// ---- POUs/OperatingModes/MBS_OperatingModes.TcPOU
FUNCTION_BLOCK MBS_OperatingModes
VAR_INPUT
	Start 			: BOOL;
	Stop			: BOOL;
	Reset			: BOOL;
	Schalter		: BOOL;
	Schrittkette_GS : BOOL;
END_VAR
VAR_OUTPUT
	A1 : BOOL; //Initialzustand
	A2 : BOOL; //Stillstand angefordert am Ende des Zyklus
//	A3 : BOOL; //Stillstand angefordert in einem bestimmten Zustand
//	A4 : BOOL; //Erhaltener Stillstand
//	A5 : BOOL; //Vorbereitung zur Wiederaufnahme nach Störung
	A6 : BOOL; //Fahrt in den Initialzustand
	F1 : BOOL; //Normalbetrieb
//	F2 : BOOL; //Anfahren
//	F3 : BOOL; //Abfahren
	F4 : BOOL; //Handbetrieb
//	F5 : BOOL; //Schrittbetrieb
//	F6 : BOOL; //Testbetrieb
//	D1 : BOOL; //Not-Aus
//	D2 : BOOL; //DIagnose und Störbehandlung
//	D3 : BOOL; //Produktion trotz Störung
END_VAR
VAR
	bFirstScan : BOOL := TRUE;	
	
	RS_InitialState: RS;	
	RS_InitialDrive: RS;
	RS_ManualOperationMode: RS;
	RS_AutomaticOperationMode: RS;
	RS_CycleEnded: RS;

	R_TRIG_Manual: R_TRIG;
	R_TRIG_Automatic: R_TRIG;
	R_TRIG_InitialDrive: R_TRIG;
	R_TRIG_CycleEnded: R_TRIG;
	R_TRIG_Init: R_TRIG;
END_VAR

R_TRIG_InitialDrive(CLK := RS_InitialDrive);
R_TRIG_CycleEnded(CLK := RS_CycleEnded);
R_TRIG_Manual(CLK := RS_ManualOperationMode);
R_TRIG_Automatic(CLK := RS_AutomaticOperationMode);
RS_InitialState(SET := ((((R_TRIG_InitialDrive.Q) AND (Schrittkette_GS))) OR (((R_TRIG_CycleEnded.Q) AND (Schrittkette_GS)))), RESET1 := ((R_TRIG_Manual.Q) OR (R_TRIG_Automatic.Q)));
A1 := RS_InitialState.Q1;
RS_ManualOperationMode(SET := ((Schalter) AND (A1) AND (Reset)), RESET1 := A6);
F4 := RS_ManualOperationMode.Q1;
R_TRIG_Manual(CLK := RS_ManualOperationMode);
R_TRIG_Init(CLK := RS_InitialState);
RS_InitialDrive(SET := ((((R_TRIG_Manual.Q) AND (((Stop) OR (NOT (Schalter)))))) OR ((bFirstScan))), RESET1 := R_TRIG_Init.Q);
A6 := RS_InitialDrive.Q1;
R_TRIG_Init(CLK := RS_InitialState);
R_TRIG_CycleEnded(CLK := RS_CycleEnded);
RS_AutomaticOperationMode(SET := ((Start) AND (R_TRIG_Init.Q) AND (NOT (Schalter))), RESET1 := R_TRIG_CycleEnded.Q);
F1 := RS_AutomaticOperationMode.Q1;
R_TRIG_Automatic(CLK := RS_AutomaticOperationMode);
R_TRIG_Init(CLK := RS_InitialState);
RS_CycleEnded(SET := ((R_TRIG_Automatic.Q) AND (((Schalter) OR (Stop)))), RESET1 := R_TRIG_Init.Q);
A2 := RS_CycleEnded.Q1;

END_FUNCTION_BLOCK

// ---- POUs/MethodenBeispiele/FB_MyOpcUaMethod.TcPOU
FUNCTION_BLOCK PUBLIC FB_MyOpcUaMethod
VAR_INPUT
	in1 : INT;
	in2 : INT;
END_VAR
VAR_OUTPUT
	result : INT;
END_VAR

{attribute 'TcRpcEnable' := '1'}
METHOD PUBLIC Multiply : INT
VAR_INPUT
	a : INT;
	b : INT;
END_VAR
Multiply := a * b;
END_METHOD

END_FUNCTION_BLOCK

// ---- POUs/MethodenBeispiele/JobMethode_Schablone.TcPOU
{attribute 'OPC.UA.DA.JobMethod' := 'JobMethode_Schablone'}
FUNCTION_BLOCK JobMethode_Schablone
VAR
	AlwaysTrue : BOOL := TRUE;
	// Used for debugging purposes to display InputArguments of method call
	MethodCall_Name : BOOL := FALSE; // used to store InputArg "MethodCall" from Start() method
	Direction_01 : BOOL := FALSE;
	Direction_02 : BOOL := FALSE;
	TS_EndschalterEntlastung : BOOL;
	callCounterStart : ULINT; // counts how many times the Start() method has been called
	callCounterCheckState : ULINT; // counts how many times the CheckState() method has been called
	callCounterAbort : ULINT; // counts how many times the Abort() method has been called
	
	// Variables to determine if a job has been started (Start() method has been called) or finished
	jobRunning : BOOL;
	jobFinished : BOOL;

	// State machine variable
	state : UDINT;
	
	//Variablen des Transport FBs
	ResetCall : BOOL := FALSE;	
	JobMethode_Name : AxisControl_MultipleInputSensors;
END_VAR
	
VAR_INPUT
	NotAusSignal: BOOL;
	LightSensor_01 : BOOL;
	LightSensor_02 : BOOL;
	TS_Endschalter_01 : BOOL;
	TS_Endschalter_02 : BOOL;
	TOF_Time_Motoransteuerung : TIME;
	TOF_Time_EndschalterEntlastung : TIME;
END_VAR

VAR_OUTPUT
	Motor_Ansteuerung01 : BOOL;
	Motor_Ansteuerung02 : BOOL;
END_VAR

JobMethode_Name(
    MethodCall := MethodCall_Name,
    NotAus_Signal := NotAusSignal,
    Direction_01 := Direction_01,
    Direction_02 := Direction_02,
    LightSensor_01 := LightSensor_01,
    LightSensor_02 := LightSensor_02,
    TS_Endschalter_01 := TS_Endschalter_01,
    AutomaticMode := _REFACTOR_,
    TS_Endschalter_02 := TS_Endschalter_02,
    TS_EndschalterEntlastung := TS_EndschalterEntlastung,
    TOF_Time_Motoransteuerung := TOF_Time_Motoransteuerung,
    TOF_Time_EndschalterEntlastung := TOF_Time_EndschalterEntlastung
);
Motor_Ansteuerung01 := JobMethode_Name.Motor_Direction01;

{attribute 'TcRpcEnable' := '1'}
METHOD Abort : HRESULT
VAR_INPUT
	hdl : UDINT; // Do not change, used by server.
END_VAR
callCounterAbort := callCounterAbort + 1;
END_METHOD

{attribute 'TcRpcEnable' := '1'}
METHOD CheckState : HRESULT
VAR_INPUT
	hdl : UDINT; // Do not change, used by server.
END_VAR
VAR_OUTPUT
	bBusy : BOOL; // Do not change. Used by server to find out if the job is finished
	
	// List of OutputArguments for OPC UA method, may be customized
	State : BOOL; // Abgeschlossener MethodCall
	MethodCall: BOOL; //Input Recall
END_VAR
callCounterCheckState := callCounterCheckState + 1;
IF NOT jobFinished THEN
	bBusy := TRUE; // job is not finished yet
	CheckState := 0; // no error
ELSE
	bBusy := FALSE; // job is finished
	CheckState := 0; // done, no error occured during execution (OPC UA StatusCode "GOOD")
	jobFinished := FALSE;
	State := ResetCall;
	MethodCall := MethodCall_Name;
END_IF
END_METHOD

{attribute 'TcRpcEnable' := '1'}
METHOD Start : HRESULT
VAR_INPUT
	// List of InputArguments for OPC UA method, may be customized
	MethodCall : BOOL; // some description
	DirectionPointA : BOOL;
	DirectionPointB : BOOL;
	EndschalterEntlastung : BOOL;	
END_VAR
VAR_OUTPUT
	hdl : UDINT; // Do not change, used by server.
END_VAR
callCounterStart := callCounterStart + 1;

MethodCall_Name := MethodCall;
DirectionPointA := Direction_01;
DirectionPointB := Direction_02;
EndschalterEntlastung := EndschalterEntlastung;

IF DirectionPointA := TRUE THEN
	DirectionPointB := FALSE;
END_IF

IF DirectionPointB := TRUE THEN
	DirectionPointA := FALSE;
END_IF

jobRunning := TRUE;
Start := 0; // no error occured, e.g. while parsing the input arguments (0 = OPC UA StatusCode "GOOD")
END_METHOD

END_FUNCTION_BLOCK

// ---- POUs/Moduls/SST_Skills/SST_CB_AS_HorizontalMove.TcPOU
{attribute 'OPC.UA.DA.JobMethod' := 'JobMethode_HorizontalMove'}
FUNCTION_BLOCK SST_CB_AS_HorizontalMove
VAR
	AlwaysTrue : BOOL := TRUE;
	// Used for debugging purposes to display InputArguments of method call
	MethodCall_HorizontalMove : BOOL := FALSE; // used to store InputArg "MethodCall" from Start() method
	ResetMethodCall : BOOL := FALSE;	
	DirectionHorizontal : STRING;
//	TS_EndschalterEntlastung : BOOL;
	callCounterStart : ULINT; // counts how many times the Start() method has been called
	callCounterCheckState : ULINT; // counts how many times the CheckState() method has been called
	callCounterAbort : ULINT; // counts how many times the Abort() method has been called
	
	// Variables to determine if a job has been started (Start() method has been called) or finished
	jobRunning : BOOL;
	jobFinished : BOOL;

	// State machine variable
	state : UDINT;
	
	//Variablen des Transport FBs
	SST_CB_HorizontalMove : AxisControl_MultipleInputSensors;
END_VAR
	
VAR_INPUT
	ESS: BOOL;
	LightSensor_01 : BOOL;
	LightSensor_02 : BOOL;
	TOF_Time_Motoransteuerung : TIME;
	AutomaticMode : BOOL;
END_VAR

VAR_OUTPUT
	DO_MovingConveyorBelt : BOOL;
END_VAR

SST_CB_HorizontalMove(
    MethodCall := MethodCall_HorizontalMove,
    EmergencyStopSignal := ESS,
    Direction := DirectionHorizontal,
    InitStateDrive_Input := ,
    DI01 := LightSensor_01,
    DI02 := LightSensor_02,
    TouchSensorRelief := ,
    TOF_Time_MotorControl := TOF_Time_Motoransteuerung,
    TOF_Time_TouchSensorRelief := ,
    OperatingMode := AutomaticMode
);
DO_MovingConveyorBelt := SST_CB_HorizontalMove.DigitalOutputControl_01;

{attribute 'TcRpcEnable' := '1'}
METHOD Abort : HRESULT
VAR_INPUT
	hdl : UDINT; // Do not change, used by server.
END_VAR
callCounterAbort := callCounterAbort + 1;
END_METHOD

{attribute 'TcRpcEnable' := '1'}
METHOD CheckState : HRESULT
VAR_INPUT
	hdl : UDINT; // Do not change, used by server.
END_VAR
VAR_OUTPUT
	bBusy : BOOL; // Do not change. Used by server to find out if the job is finished
	
	// List of OutputArguments for OPC UA method, may be customized
	State : BOOL; // Abgeschlossener MethodCall
	MethodCall: BOOL; //Input Recall
END_VAR
callCounterCheckState := callCounterCheckState + 1;
IF NOT jobFinished THEN
	bBusy := TRUE; // job is not finished yet
	CheckState := 0; // no error
ELSE
	bBusy := FALSE; // job is finished
	CheckState := 0; // done, no error occured during execution (OPC UA StatusCode "GOOD")
	jobFinished := FALSE;
	State := ResetMethodCall;
	MethodCall := MethodCall_HorizontalMove;
END_IF
END_METHOD

{attribute 'TcRpcEnable' := '1'}
METHOD Start : HRESULT
VAR_INPUT
	// List of InputArguments for OPC UA method, may be customized
	MethodCall : BOOL; // some description
	DirectionPoint : STRING;
END_VAR
VAR_OUTPUT
	hdl : UDINT; // Do not change, used by server.
END_VAR
callCounterStart := callCounterStart + 1;

MethodCall_HorizontalMove := MethodCall;
DirectionHorizontal := DirectionPoint;

jobRunning := TRUE;
Start := 0; // no error occured, e.g. while parsing the input arguments (0 = OPC UA StatusCode "GOOD")
END_METHOD

END_FUNCTION_BLOCK

// ---- POUs/Moduls/SST_Skills/SST_CS_AS_ColorDetection.TcPOU
{attribute 'OPC.UA.DA.JobMethod' := 'JobMethode_ColorDetection'}
FUNCTION_BLOCK SST_CS_AS_ColorDetection
VAR
	AlwaysTrue : BOOL := TRUE;
	// Used for debugging purposes to display InputArguments of method call
	MethodCall_ColorDetection : BOOL := FALSE; // used to store InputArg "MethodCall" from Start() method
	callCounterStart : ULINT; // counts how many times the Start() method has been called
	callCounterCheckState : ULINT; // counts how many times the CheckState() method has been called
	callCounterAbort : ULINT; // counts how many times the Abort() method has been called
	
	// Variables to determine if a job has been started (Start() method has been called) or finished
	jobRunning : BOOL;
	jobFinished : BOOL;

	// State machine variable
	state : UDINT;
	
	//Variablen des Transport FBs
	ResetCall : BOOL := FALSE;	
	SST_Auto_ColorDetection : AutomaticColorDetection_nichtfertig;
	
	//Farbcodes
	ColorCode1 : INT ;
	ColorCode2 : INT ;
	ColorCode3 : INT ;
END_VAR
	
VAR_INPUT
	Color_Sensor : INT;
END_VAR

VAR_OUTPUT
 Color_White : BOOL;
 Color_Red : BOOL;
 Color_Blue : BOOL;
END_VAR

SST_Auto_ColorDetection(ColorSensor := Color_Sensor, ColorCode_1 := ColorCode1, ColorCode_2 := ColorCode2, ColorCode_3 := ColorCode3);
Color_White := SST_Auto_ColorDetection.Color_1;

{attribute 'TcRpcEnable' := '1'}
METHOD Abort : HRESULT
VAR_INPUT
	hdl : UDINT; // Do not change, used by server.
END_VAR
callCounterAbort := callCounterAbort + 1;
END_METHOD

{attribute 'TcRpcEnable' := '1'}
METHOD CheckState : HRESULT
VAR_INPUT
	hdl : UDINT; // Do not change, used by server.
END_VAR
VAR_OUTPUT
	bBusy : BOOL; // Do not change. Used by server to find out if the job is finished
	
	// List of OutputArguments for OPC UA method, may be customized
	State : BOOL; // Abgeschlossener MethodCall
	MethodCall: BOOL; //Input Recall
END_VAR
callCounterCheckState := callCounterCheckState + 1;
IF NOT jobFinished THEN
	bBusy := TRUE; // job is not finished yet
	CheckState := 0; // no error
ELSE
	bBusy := FALSE; // job is finished
	CheckState := 0; // done, no error occured during execution (OPC UA StatusCode "GOOD")
	jobFinished := FALSE;
	State := ResetCall;
	MethodCall := MethodCall_ColorDetection;
END_IF
END_METHOD

{attribute 'TcRpcEnable' := '1'}
METHOD Start : HRESULT
VAR_INPUT
	// List of InputArguments for OPC UA method, may be customized
	MethodCall : BOOL; // some description
	DirectionPointA : BOOL;
	DirectionPointB : BOOL;
	EndschalterEntlastung : BOOL;	
END_VAR
VAR_OUTPUT
	hdl : UDINT; // Do not change, used by server.
END_VAR
callCounterStart := callCounterStart + 1;

MethodCall_ColorDetection := MethodCall;

jobRunning := TRUE;
Start := 0; // no error occured, e.g. while parsing the input arguments (0 = OPC UA StatusCode "GOOD")
END_METHOD

END_FUNCTION_BLOCK

// ---- POUs/Moduls/SST_Skills/SST_PD_AS_HorizontalMove.TcPOU
{attribute 'OPC.UA.DA.JobMethod' := 'JobMethode_CompressorControl'}
FUNCTION_BLOCK SST_PD_AS_HorizontalMove
VAR
	AlwaysTrue : BOOL := TRUE;
	// Used for debugging purposes to display InputArguments of method call
	MethodCall_CompressorControl : BOOL := FALSE; // used to store InputArg "MethodCall" from Start() method
	ResetMethodCall : BOOL := FALSE;
	DestinationHorizontal : STRING;
	callCounterStart : ULINT; // counts how many times the Start() method has been called
	callCounterCheckState : ULINT; // counts how many times the CheckState() method has been called
	callCounterAbort : ULINT; // counts how many times the Abort() method has been called
	
	// Variables to determine if a job has been started (Start() method has been called) or finished
	jobRunning : BOOL;
	jobFinished : BOOL;

	// State machine variable
	state : UDINT;
	
	//Variablen des Transport FBs
	
	MBS_VSG_HorizontalMove : CompressorControl;
END_VAR
	
VAR_INPUT
	ESS: BOOL;
	LightSensor_01 : BOOL;
	LightSensor_02 : BOOL;
	PowerOnDelay_Compressor : TIME;
	PowerOnDelay_Valve : TIME;
	AutomaticMode : BOOL;
END_VAR

VAR_OUTPUT
	DO_ControlCompressorPD_01 : BOOL;
	DO_ControlValvePD_02 : BOOL;
END_VAR

MBS_VSG_HorizontalMove(
    MethodCall := MethodCall_CompressorControl,
    EmergencyStopSignal := ESS,
    Destination := DestinationHorizontal,
    InitStateDrive_Input := ,
    DI01 := LightSensor_01,
    DI02 := LightSensor_02,
    DI03_EncoderStart01 := ,
    DI04_EncoderStart02 := ,
    DI05_EncoderStart03 := ,
    DI06_EncoderStart04 := ,
    DI07_EncoderStart05 := ,
    DI08_EncoderStart06 := ,
    DI09_EncoderTarget01 := ,
    DI10_EncoderTarget02 := ,
    DI11_EncoderTarget03 := ,
    DI12_EncoderTarget04 := ,
    DI13_EncoderTarget05 := ,
    DI14_EncoderTarget06 := ,
    PowerOFF_SelfSet := ,
    TON_Time_PowerOFFSelfSet := ,
    TON_Time_Compressor := PowerOnDelay_Compressor,
    TON_Time_Valve := PowerOnDelay_Valve,
    OperatingMode := AutomaticMode
);
DO_ControlCompressorPD_01 := MBS_VSG_HorizontalMove.DigitalOutputControl_01;

{attribute 'TcRpcEnable' := '1'}
METHOD Abort : HRESULT
VAR_INPUT
	hdl : UDINT; // Do not change, used by server.
END_VAR
callCounterAbort := callCounterAbort + 1;
END_METHOD

{attribute 'TcRpcEnable' := '1'}
METHOD CheckState : HRESULT
VAR_INPUT
	hdl : UDINT; // Do not change, used by server.
END_VAR
VAR_OUTPUT
	bBusy : BOOL; // Do not change. Used by server to find out if the job is finished
	
	// List of OutputArguments for OPC UA method, may be customized
	State : BOOL; // Abgeschlossener MethodCall
	MethodCall: BOOL; //Input Recall
END_VAR
callCounterCheckState := callCounterCheckState + 1;
IF NOT jobFinished THEN
	bBusy := TRUE; // job is not finished yet
	CheckState := 0; // no error
ELSE
	bBusy := FALSE; // job is finished
	CheckState := 0; // done, no error occured during execution (OPC UA StatusCode "GOOD")
	jobFinished := FALSE;
	State := ResetMethodCall;
	MethodCall := MethodCall_CompressorControl;
END_IF
END_METHOD

{attribute 'TcRpcEnable' := '1'}
METHOD Start : HRESULT
VAR_INPUT
	// List of InputArguments for OPC UA method, may be customized
	MethodCall : BOOL; // some description
	DestinationPoint : STRING;	
END_VAR
VAR_OUTPUT
	hdl : UDINT; // Do not change, used by server.
END_VAR
callCounterStart := callCounterStart + 1;

MethodCall_CompressorControl := MethodCall;
DestinationHorizontal := DestinationPoint;

jobRunning := TRUE;
Start := 0; // no error occured, e.g. while parsing the input arguments (0 = OPC UA StatusCode "GOOD")
END_METHOD

END_FUNCTION_BLOCK

// ---- POUs/OperatingModes/SST_OperatingModes.TcPOU
FUNCTION_BLOCK SST_OperatingModes
VAR_INPUT
	Start 			: BOOL;
	Stop			: BOOL;
	Reset			: BOOL;
	Schalter		: BOOL;
	Schrittkette_GS : BOOL;
END_VAR
VAR_OUTPUT
	A1 : BOOL; //Initialzustand
	A2 : BOOL; //Stillstand angefordert am Ende des Zyklus
//	A3 : BOOL; //Stillstand angefordert in einem bestimmten Zustand
//	A4 : BOOL; //Erhaltener Stillstand
//	A5 : BOOL; //Vorbereitung zur Wiederaufnahme nach Störung
	A6 : BOOL; //Fahrt in den Initialzustand
	F1 : BOOL; //Normalbetrieb
//	F2 : BOOL; //Anfahren
//	F3 : BOOL; //Abfahren
	F4 : BOOL; //Handbetrieb
//	F5 : BOOL; //Schrittbetrieb
//	F6 : BOOL; //Testbetrieb
//	D1 : BOOL; //Not-Aus
//	D2 : BOOL; //DIagnose und Störbehandlung
//	D3 : BOOL; //Produktion trotz Störung
END_VAR
VAR
	bFirstScan : BOOL := TRUE;	
	
	RS_InitialState: RS;	
	RS_InitialDrive: RS;
	RS_ManualOperationMode: RS;
	RS_AutomaticOperationMode: RS;
	RS_CycleEnded: RS;

	R_TRIG_Manual: R_TRIG;
	R_TRIG_Automatic: R_TRIG;
	R_TRIG_InitialDrive: R_TRIG;
	R_TRIG_CycleEnded: R_TRIG;
	R_TRIG_Init: R_TRIG;
END_VAR

R_TRIG_InitialDrive(CLK := RS_InitialDrive);
R_TRIG_CycleEnded(CLK := RS_CycleEnded);
R_TRIG_Manual(CLK := RS_ManualOperationMode);
R_TRIG_Automatic(CLK := RS_AutomaticOperationMode);
RS_InitialState(SET := ((((R_TRIG_InitialDrive.Q) AND (Schrittkette_GS))) OR (((R_TRIG_CycleEnded.Q) AND (Schrittkette_GS)))), RESET1 := ((R_TRIG_Manual.Q) OR (R_TRIG_Automatic.Q)));
A1 := RS_InitialState.Q1;
RS_ManualOperationMode(SET := ((Schalter) AND (A1) AND (Reset)), RESET1 := A6);
F4 := RS_ManualOperationMode.Q1;
R_TRIG_Manual(CLK := RS_ManualOperationMode);
R_TRIG_Init(CLK := RS_InitialState);
RS_InitialDrive(SET := ((((R_TRIG_Manual.Q) AND (((Stop) OR (NOT (Schalter)))))) OR ((bFirstScan))), RESET1 := R_TRIG_Init.Q);
A6 := RS_InitialDrive.Q1;
R_TRIG_Init(CLK := RS_InitialState);
R_TRIG_CycleEnded(CLK := RS_CycleEnded);
RS_AutomaticOperationMode(SET := ((Start) AND (R_TRIG_Init.Q) AND (NOT (Schalter))), RESET1 := R_TRIG_CycleEnded.Q);
F1 := RS_AutomaticOperationMode.Q1;
R_TRIG_Automatic(CLK := RS_AutomaticOperationMode);
R_TRIG_Init(CLK := RS_InitialState);
RS_CycleEnded(SET := ((R_TRIG_Automatic.Q) AND (((Schalter) OR (Stop)))), RESET1 := R_TRIG_Init.Q);
A2 := RS_CycleEnded.Q1;

END_FUNCTION_BLOCK

// ---- POUs/OperatingModes/VSG_OperatingModes_alt.TcPOU
FUNCTION_BLOCK VSG_OperatingModes_alt
VAR_INPUT
	Start 			: BOOL;
	Stop			: BOOL;
	Reset			: BOOL;
	Schalter		: BOOL;
	Schrittkette_GS : BOOL;
END_VAR
VAR_OUTPUT
	A1 : BOOL; //Initialzustand
	A2 : BOOL; //Stillstand angefordert am Ende des Zyklus
//	A3 : BOOL; //Stillstand angefordert in einem bestimmten Zustand
//	A4 : BOOL; //Erhaltener Stillstand
//	A5 : BOOL; //Vorbereitung zur Wiederaufnahme nach Störung
	A6 : BOOL; //Fahrt in den Initialzustand
	F1 : BOOL; //Normalbetrieb
//	F2 : BOOL; //Anfahren
//	F3 : BOOL; //Abfahren
	F4 : BOOL; //Handbetrieb
//	F5 : BOOL; //Schrittbetrieb
//	F6 : BOOL; //Testbetrieb
//	D1 : BOOL; //Not-Aus
//	D2 : BOOL; //DIagnose und Störbehandlung
//	D3 : BOOL; //Produktion trotz Störung
END_VAR
VAR
	bFirstScan : BOOL := TRUE;	
	
	RS_InitialState: RS;	
	RS_InitialDrive: RS;
	RS_ManualOperationMode: RS;
	RS_AutomaticOperationMode: RS;
	RS_CycleEnded: RS;

	R_TRIG_Manual: R_TRIG;
	R_TRIG_Automatic: R_TRIG;
	R_TRIG_InitialDrive: R_TRIG;
	R_TRIG_CycleEnded: R_TRIG;
	R_TRIG_Init: R_TRIG;
END_VAR
VAR // added by the converter: edge detectors and wires of the graphical bodies
    _w1 : BOOL;
END_VAR

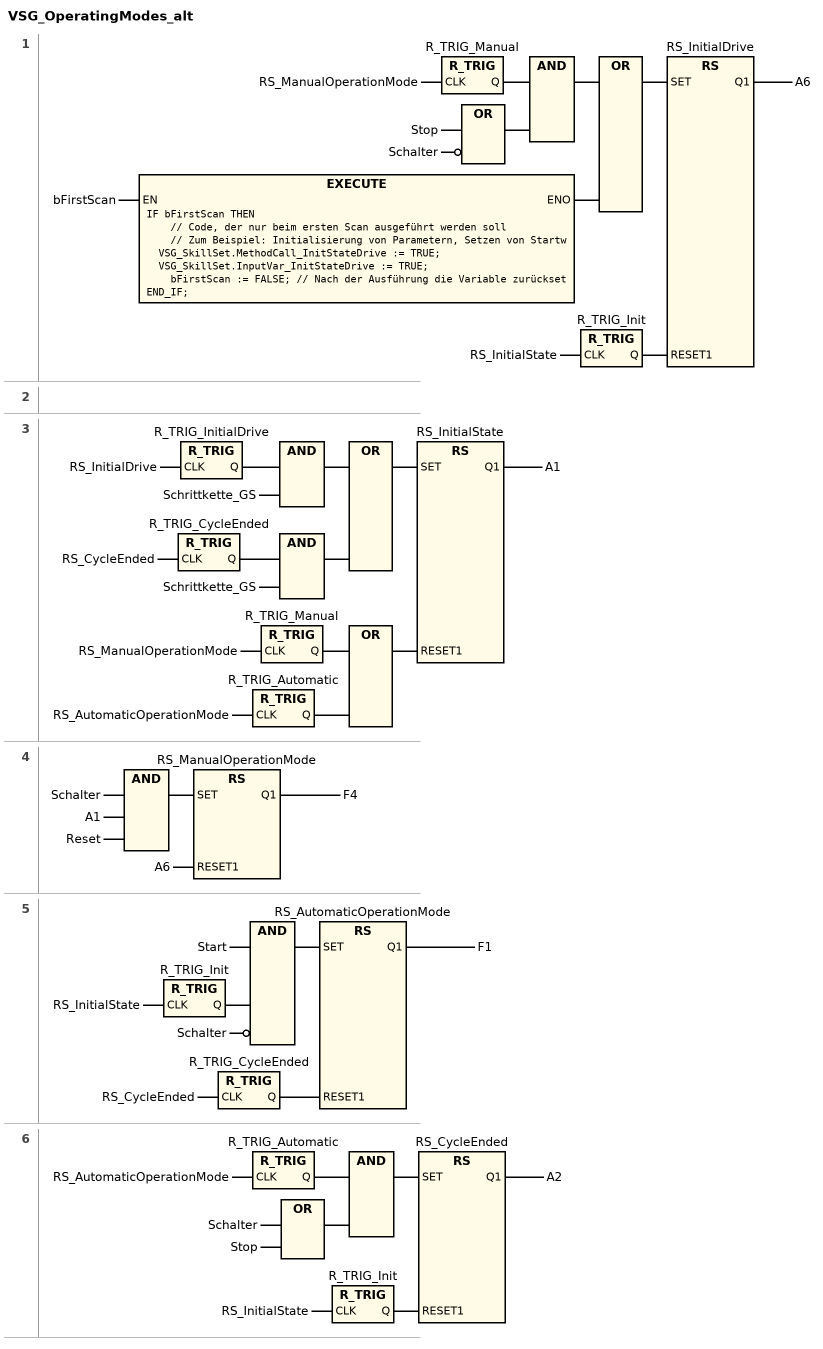
// NETWORK 1
R_TRIG_Manual(CLK := RS_ManualOperationMode); // R_TRIG
_w1 := bFirstScan;
IF _w1 THEN
    IF bFirstScan THEN
        // Code, der nur beim ersten Scan ausgeführt werden soll
        // Zum Beispiel: Initialisierung von Parametern, Setzen von Startwerten etc.
    	VSG_SkillSet.MethodCall_InitStateDrive := TRUE;
    	VSG_SkillSet.InputVar_InitStateDrive := TRUE;
        bFirstScan := FALSE; // Nach der Ausführung die Variable zurücksetzen
    END_IF;
END_IF
R_TRIG_Init(CLK := RS_InitialState); // R_TRIG
RS_InitialDrive(SET := R_TRIG_Manual.Q AND (Stop OR NOT Schalter) OR _w1, RESET1 := R_TRIG_Init.Q); // RS
A6 := RS_InitialDrive.Q1;

// NETWORK 2

// NETWORK 3
R_TRIG_InitialDrive(CLK := RS_InitialDrive); // R_TRIG
R_TRIG_CycleEnded(CLK := RS_CycleEnded); // R_TRIG
R_TRIG_Manual(CLK := RS_ManualOperationMode); // R_TRIG
R_TRIG_Automatic(CLK := RS_AutomaticOperationMode); // R_TRIG
RS_InitialState(SET := R_TRIG_InitialDrive.Q AND Schrittkette_GS OR R_TRIG_CycleEnded.Q AND Schrittkette_GS, RESET1 := R_TRIG_Manual.Q OR R_TRIG_Automatic.Q); // RS
A1 := RS_InitialState.Q1;

// NETWORK 4
RS_ManualOperationMode(SET := Schalter AND A1 AND Reset, RESET1 := A6); // RS
F4 := RS_ManualOperationMode.Q1;

// NETWORK 5
R_TRIG_Init(CLK := RS_InitialState); // R_TRIG
R_TRIG_CycleEnded(CLK := RS_CycleEnded); // R_TRIG
RS_AutomaticOperationMode(SET := Start AND R_TRIG_Init.Q AND NOT Schalter, RESET1 := R_TRIG_CycleEnded.Q); // RS
F1 := RS_AutomaticOperationMode.Q1;

// NETWORK 6
R_TRIG_Automatic(CLK := RS_AutomaticOperationMode); // R_TRIG
R_TRIG_Init(CLK := RS_InitialState); // R_TRIG
RS_CycleEnded(SET := R_TRIG_Automatic.Q AND (Schalter OR Stop), RESET1 := R_TRIG_Init.Q); // RS
A2 := RS_CycleEnded.Q1;

END_FUNCTION_BLOCK

// ---- POUs/SST_SkillSet.TcPOU
PROGRAM SST_SkillSet
VAR
//Farbscanner- & Sortiertanlage Skills
	//ColorSensor Skills
	{attribute 'OPC.UA.DA':= '1'}
	SST_AutomaticColorDetection : SST_CS_AS_ColorDetection;
	
	//ConveyorBelt Skills
	{attribute 'OPC.UA.DA':= '1'}
	SST_ConveyorBeltMoveHorizontal_ToPD01 : SST_CB_AS_HorizontalMove;
	{attribute 'OPC.UA.DA':= '1'}
	SST_ConveyorBeltMoveHorizontal_ToPD02 : SST_CB_AS_HorizontalMove;
	{attribute 'OPC.UA.DA':= '1'}
	SST_ConveyorBeltMoveHorizontal_ToPD03 : SST_CB_AS_HorizontalMove;
	{attribute 'OPC.UA.DA':= '1'}
	SST_ConveyorBeltMoveHorizontal_TillEnd : SST_CB_AS_HorizontalMove;
	
	//PushingDeviceStation Skills
	{attribute 'OPC.UA.DA':= '1'}
	SST_PD01_HorizontalMove : SST_PD_AS_HorizontalMove;
	{attribute 'OPC.UA.DA':= '1'}
	SST_PD02_HorizontalMove : SST_PD_AS_HorizontalMove;
	{attribute 'OPC.UA.DA':= '1'}
	SST_PD03_HorizontalMove : SST_PD_AS_HorizontalMove;
	
	//Organisation FBs
	SST_OperatingModes : SST_OperatingModes;
	SST_ControlOfOutputs : SST_ControlOfOutputs;
	
	//InitialStateDrives	
	SST_PD_InitStateDrive: SST_PD_InitialStateDrive;

//Variablen zur Outputsteuerung
	//Output-Variablen der Komponente ConveyorBelt	
	CB_MoveForwardToPD01: BOOL;
	CB_MoveForwardToPD02: BOOL;
	CB_MoveForwardToPD03: BOOL;
	CB_MoveForwardTillEnd: BOOL;
	
	//Output-Variablen der Komponente PushingDevice
	PD01_Compressor : BOOL;
	PD02_Compressor : BOOL;
	PD03_Compressor : BOOL;
	PD01_Valve : BOOL;
	PD02_Valve : BOOL;
	PD03_Valve : BOOL;	
	
	//Output-Variablen für Init-Fahrt
	Init_PD01_Compressor : BOOL;
	Init_PD02_Compressor : BOOL;
	Init_PD03_Compressor : BOOL;
	Init_PD01_Valve : BOOL;
	Init_PD02_Valve : BOOL;
	Init_PD03_Valve : BOOL;
	
//Variablensetzung: Sollte später über SkillOA eingesetzt werden ODER Hard in SPS codiert (Diskussionspunkt)
	ResetButton: BOOL;
	StartButton: BOOL;
	ConfirmationButton: BOOL;

//Time Constraints
	TOF_Time_TransportPD01 : TIME;
	TOF_Time_TransportPD02 : TIME;
	TOF_Time_TransportPD03 : TIME;
	TON_Time_PD01Compressor : TIME;
	TON_Time_PD02Compressor : TIME;
	TON_Time_PD03Compressor : TIME;
	TON_Time_PD01Valve : TIME;
	TON_Time_PD02Valve : TIME;
	TON_Time_PD03Valve : TIME;
	TON_Time_PowerOFFSelfSet : TIME := T#150MS;
	
//Variable Values for InitialStateDrive
	MethodCall_InitStateDrive	: BOOL;
	InputVar_InitStateDrive		: BOOL;

END_VAR

SST_OperatingModes(
    Start := StartButton,
    Stop := ((GVL.diNotAus_Kanal_A) AND (GVL.diNotAus_Kanal_B)),
    Reset := ResetButton,
    Schalter := ConfirmationButton,
    Schrittkette_GS := (((SST_PD_InitStateDrive.ResetMethodCallMovePD01) AND (SST_PD_InitStateDrive.ResetMethodCallMovePD02) AND (SST_PD_InitStateDrive.ResetMethodCallMovePD03)))
);
SST_ControlOfOutputs(
    F4 := SST_OperatingModes.F4,
    F1 := SST_OperatingModes.F1,
    A2 := SST_OperatingModes.A2,
    A1 := SST_OperatingModes.A1,
    A6 := SST_OperatingModes.A6,
    Start := SST_OperatingModes.Start,
    CB_MoveForwardToPD01 := CB_MoveForwardToPD01,
    CB_MoveForwardToPD02 := CB_MoveForwardToPD02,
    CB_MoveForwardToPD03 := CB_MoveForwardToPD03,
    CB_MoveForwardTillEnd := CB_MoveForwardTillEnd,
    PD01_Compressor := PD01_Compressor,
    PD02_Compressor := PD02_Compressor,
    PD03_Compressor := PD03_Compressor,
    PD01_Valve := PD01_Valve,
    PD02_Valve := PD02_Valve,
    PD03_Valve := PD03_Valve,
    Init_PD01_Compressor := Init_PD01_Compressor,
    Init_PD02_Compressor := Init_PD02_Compressor,
    Init_PD03_Compressor := Init_PD03_Compressor,
    Init_PD01_Valve := Init_PD01_Valve,
    Init_PD02_Valve := Init_PD02_Valve,
    Init_PD03_Valve := Init_PD03_Valve
);
GVL_SST.SST_MOT_Foerderband := SST_ControlOfOutputs.ConveyorBeltForward;
SST_PD_InitStateDrive(
    MethodCall_InitDrive := MethodCall_InitStateDrive,
    ESS := ((GVL.diNotAus_Kanal_A) AND (GVL.diNotAus_Kanal_B)),
    InputInitialStateDrive := InputVar_InitStateDrive,
    TON_Time_PowerOFFSelfSet := TON_Time_PowerOFFSelfSet,
    InitDriveMode := SST_OperatingModes.A6
);
Init_PD01_Compressor := SST_PD_InitStateDrive.MotorControl_PD01_Compressor;
SST_AutomaticColorDetection(Color_Sensor := );
 := SST_AutomaticColorDetection.Color_White;
SST_ConveyorBeltMoveHorizontal_ToPD01(
    ESS := ((GVL.diNotAus_Kanal_A) AND (GVL.diNotAus_Kanal_B)),
    LightSensor_01 := GVL_SST.SST_LS_Eingang,
    LightSensor_02 := GVL_SST.SST_LS_nach_Farbsensor,
    TOF_Time_Motoransteuerung := TOF_Time_TransportPD01,
    AutomaticMode := SST_OperatingModes.A6
);
CB_MoveForwardToPD01 := SST_ConveyorBeltMoveHorizontal_ToPD01.DO_MovingConveyorBelt;
SST_ConveyorBeltMoveHorizontal_ToPD02(
    ESS := ((GVL.diNotAus_Kanal_A) AND (GVL.diNotAus_Kanal_B)),
    LightSensor_01 := GVL_SST.SST_LS_Eingang,
    LightSensor_02 := GVL_SST.SST_LS_nach_Farbsensor,
    TOF_Time_Motoransteuerung := TOF_Time_TransportPD02,
    AutomaticMode := SST_OperatingModes.A6
);
CB_MoveForwardToPD02 := SST_ConveyorBeltMoveHorizontal_ToPD02.DO_MovingConveyorBelt;
SST_ConveyorBeltMoveHorizontal_ToPD03(
    ESS := ((GVL.diNotAus_Kanal_A) AND (GVL.diNotAus_Kanal_B)),
    LightSensor_01 := GVL_SST.SST_LS_Eingang,
    LightSensor_02 := GVL_SST.SST_LS_nach_Farbsensor,
    TOF_Time_Motoransteuerung := TOF_Time_TransportPD03,
    AutomaticMode := SST_OperatingModes.A6
);
CB_MoveForwardToPD03 := SST_ConveyorBeltMoveHorizontal_ToPD03.DO_MovingConveyorBelt;
SST_ConveyorBeltMoveHorizontal_TillEnd(
    ESS := ((GVL.diNotAus_Kanal_A) AND (GVL.diNotAus_Kanal_B)),
    LightSensor_01 := GVL_SST.SST_LS_Eingang,
    LightSensor_02 := GVL_SST.SST_LS_nach_Farbsensor,
    TOF_Time_Motoransteuerung := ,
    AutomaticMode := SST_OperatingModes.A6
);
CB_MoveForwardTillEnd := SST_ConveyorBeltMoveHorizontal_TillEnd.DO_MovingConveyorBelt;
SST_PD01_HorizontalMove(
    ESS := ((GVL.diNotAus_Kanal_A) AND (GVL.diNotAus_Kanal_B)),
    LightSensor_01 := GVL_SST.SST_LS_nach_Farbsensor,
    LightSensor_02 := GVL_SST.SST_LS_weiss,
    PowerOnDelay_Compressor := TON_Time_PD01Compressor,
    PowerOnDelay_Valve := TON_Time_PD01Valve,
    AutomaticMode := SST_OperatingModes.A6
);
PD01_Compressor := SST_PD01_HorizontalMove.DO_ControlCompressorPD_01;
SST_PD02_HorizontalMove(
    ESS := ((GVL.diNotAus_Kanal_A) AND (GVL.diNotAus_Kanal_B)),
    LightSensor_01 := GVL_SST.SST_LS_nach_Farbsensor,
    LightSensor_02 := GVL_SST.SST_LS_rot,
    PowerOnDelay_Compressor := TON_Time_PD02Compressor,
    PowerOnDelay_Valve := TON_Time_PD02Valve,
    AutomaticMode := SST_OperatingModes.A6
);
PD02_Compressor := SST_PD02_HorizontalMove.DO_ControlCompressorPD_01;
SST_PD03_HorizontalMove(
    ESS := ((GVL.diNotAus_Kanal_A) AND (GVL.diNotAus_Kanal_B)),
    LightSensor_01 := GVL_SST.SST_LS_nach_Farbsensor,
    LightSensor_02 := GVL_SST.SST_LS_blau,
    PowerOnDelay_Compressor := TON_Time_PD03Compressor,
    PowerOnDelay_Valve := TON_Time_PD03Valve,
    AutomaticMode := SST_OperatingModes.A6
);
PD03_Compressor := SST_PD03_HorizontalMove.DO_ControlCompressorPD_01;

END_PROGRAM
